Yaskawa INFORM job: WELDING-FRONT-ST-1.JBI

/JOB
//NAME WELDING-FRONT-ST-1
//POS
///NPOS 0,0,0,0,0,0
//INST
///DATE 2018/09/25 14:23
///ATTR SC,RW
NOP
'***** CMF 100 sensor
IFTHEN D005=8
	 CALL JOB:WELDING-CMF100-ST1-FRONT
ENDIF
'***** F........ sensors
IFTHEN D005=4
	 CALL JOB:WELDING-F-SENSORS-FRONT-ST1
ENDIF
END
